TYPE ST_Timer :
STRUCT
	bTimerStat : BOOL;
	bTimerOut : BOOL;
	tTimeElapsed : TIME;
	tTimer : TIME;
END_STRUCT
END_TYPE

(* stored: Version 1.1.0.1, ProductVersion 3.1.4024.12
   DUT ST_Timer: Id {c2d7c26c-abbc-42a8-9754-10f09f25fcee} *)
